Fanuc KAREL source: ke00004.KL

-- PROVISIONAL review KL for V770-1; original PC SHA256 ff6959ad9339e15064ab760131ba5b06a98eea07753a15567df7aa2a1e9fd8d1
-- Incomplete behavior may be omitted. Consult companion uncertainty JSON. Do not deploy.
PROGRAM KE00004
%NOLOCKGROUP
BEGIN
  -- UNRESOLVED_PC offsets 5-12; opcodes 9D,23
  -- UNRESOLVED_PC offsets 17-29; opcodes 3F,75
  -- UNRESOLVED_PC offsets 34-58; opcodes 27,22,22,2A,22,31
  -- UNRESOLVED_PC offsets 63-67; opcodes 7F
END KE00004
